(* PLC project stockage, TNI-Software ControlBuild 4.00 *)
(* stored: creationDateTime 2018-09-17T17:05:16-01:00 *)

CONFIGURATION stockage
  VAR_GLOBAL
    simuperiod : REAL := 50000.0;
    taskname : STRING(50) := 'stockage.exe';
    allowpreconditions : BOOL := true;
    allowpostconditions : BOOL := true;
  END_VAR
END_CONFIGURATION
